Staubli VAL3: instruction.pjx

--- instruction.pjx ---
Parameters version=s7.5 stackSize=5000 millimeterUnit=true
Program file=find.pgx
Program file=get.pgx
Program file=getSize.pgx
Program file=getType.pgx
Program file=load.pgx
Program file=onEdit.pgx
Program file=onInsert.pgx
Program file=onProgEnd.pgx
Program file=onRun.pgx
Program file=onStart.pgx
Program file=onStop.pgx
Data file=instruction.dtx
Library alias=cycleStatus path=Disk://cycleStatus/cycleStatus.pjx

--- find.pgx ---
public program find(string& x_sItem[], bool& x_bFound[])
begin
  //
  // find one item in the list
  //
end

--- get.pgx ---
public program get(string& x_sItem[], num x_nIndex)
begin
  //
  // get one element from the list
  //
end

--- load.pgx ---
public program load(string x_sItem, num& x_nResult)
  local string l_sType
  local string l_sMessage
begin
  // load it

end

--- onInsert.pgx ---
public program onInsert(string& x_sItem[])
  local string l_sItem
begin
  //
  // compose the string
  // call getType(l_sItem)
  // x_sItem=l_sItem+" ???"
  //
end

--- onProgEnd.pgx ---
public program onProgEnd(string& x_sItem[])
begin
  //
  // Done, when one program has finished
  //
end

--- onRun.pgx ---
public program onRun(string& x_sItem[])
begin
  //
  // Done, when you execute it
  //
end

--- onStop.pgx ---
public program onStop(string& x_sItem[])
begin
  //
  // Done after a stop
  //
end
